FUNCTION_BLOCK Conveyor1HmiIProv (* Conveyor HMI Interface publish *)
  (* Standard: 61499-2 *)
  (* Version 0.2, 2003-12-05, JHC, Rockwell Automation, Renamed from NEWCOMPFB. *)
  (* Version 0.1, 2002-01-08, JHC, Rockwell Automation, Added DLY FB as example. *)
  (* Version 0.0, 2000-05-27, JHC, Rockwell Automation *)
  (* Compiler header: package fb.rt.dasdA1.A2.Conveyor; *)
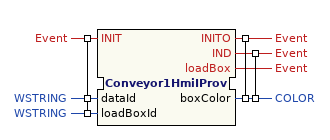
  EVENT_INPUT
    INIT WITH dataId, loadBoxId; (* Initialization Request *)
  END_EVENT
  EVENT_OUTPUT
    INITO WITH boxColor; (* Initialization Confirm *)
    IND WITH boxColor;
    loadBox;
  END_EVENT
  VAR_INPUT
    dataId : WSTRING;
    loadBoxId : WSTRING;
  END_VAR
  VAR_OUTPUT
    boxColor : COLOR;
  END_VAR
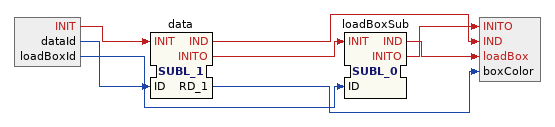
  FBS
    loadBoxSub : SUBL_0;
    data : SUBL_1;
  END_FBS
  EVENT_CONNECTIONS
    loadBoxSub.IND TO loadBox;
    INIT TO data.INIT;
    data.IND TO IND;
    data.INITO TO loadBoxSub.INIT;
    loadBoxSub.INITO TO INITO;
  END_CONNECTIONS
  DATA_CONNECTIONS
    loadBoxId TO loadBoxSub.ID;
    dataId TO data.ID;
    data.RD_1 TO boxColor;
  END_CONNECTIONS
END_FUNCTION_BLOCK
